RESOURCE_TYPE ResourceType (* Resource Type *)
  (* Standard: 61499-2 *)
  (* Version 0.1, 2003-12-05, JHC, Rockwell Automation, Renamed from NEWRESOURCE. *)
  (* Version 0.0, 2000-05-27, JHC, Rockwell Automation *)
  (* Compiler header: package fb.rt.template; *)
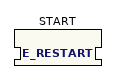
  FBS
    START : E_RESTART;
  END_FBS
END_RESOURCE_TYPE
